// TIA Portal V16 export
// export: Created 2021-07-12T14:47:20.3940069Z, ExportSetting WithDefaults, DisplayName Totally Integrated Automation Portal, DisplayVersion V16, DisplayName TIA Portal Version Control Interface, DisplayVersion V16, DisplayName TIA Portal Openness, DisplayVersion V16, DisplayName STEP 7 Professional, DisplayVersion V16, DisplayName STEP 7 Safety, DisplayVersion V16, DisplayName WinCC Professional, DisplayVersion V16
TYPE "SimaHydTO_typeHMIConnectionHmiData"
TITLE = SimaHydTO_typeHMIConnectionHmiData
// HMI interface: Data to display on HMI
// stored: IsFailsafeCompliant false
   STRUCT
      stateSubNavigation : Int;
      ActualPositionPercent : Int;   // Actual axis position in percent between MinPosition and MaxPosition
      SafetyDistanceAnimation : LReal;   // SafetyDistance in percent between MinPosition and MaxPosition
      MinPosition : LReal;   // Minimal position of axis (SW limit switch)
      MaxPosition : LReal;   // Maximal position of axis (SW limit switch)
      selectedAxis : Int;   // DB number of actual selected hydraulic axis
      selectedAxisTO : Int;   // DB/TO number of actual selected technology object
      selectedVChar : Int;   // DB number of actual selected valve characteristics
      VChar { S7_SetPoint := 'True'} : "SimaHydTO_typeHMIConnectionHmiDataVChar";   // Data storage of HMI VChar display
   END_STRUCT;
END_TYPE
